// TwinCAT 3 PLC project Twinson
// Title: Twinson
// Company: Stefan Besler
// ProjectVersion: 0.2.0.0
// ProgramVersion: 3.1.4023.0
// project tree:
//   JsonDecoder/ IJsonElement.TcIO, JsonDecoder.TcPOU, JsonElement.TcPOU, JsonElementType.TcDUT, JsonNode.TcDUT
//   JsonDecoder/_Test/ JsonDecoderTest.TcPOU
//   / ParameterList.TcGVL
//   UnitTest/ IAssertions.TcIO, IUnittest.TcIO

// ---- JsonDecoder/JsonElementType.TcDUT
{attribute 'qualified_only'}
TYPE JsonElementType :
(
  Undefined := 0,
  Strng,
  Number,
  Object,
  Arry,
  Boolean,
  Null
);
END_TYPE

// ---- JsonDecoder/JsonNode.TcDUT
TYPE JsonNode :
STRUCT
  Name : STRING;
  Next : REFERENCE TO JsonNode;
  Child : REFERENCE TO JsonNode;
  Element : REFERENCE TO JsonElement;
END_STRUCT
END_TYPE

// ---- ParameterList.TcGVL
{attribute 'qualified_only'}
VAR_GLOBAL CONSTANT
  MaxJsonKeyLength : INT := 31;
  MaxJsonAssignments : INT := 200;
END_VAR

// ---- JsonDecoder/IJsonElement.TcIO
INTERFACE IJsonElement

METHOD AsString : STRING
END_METHOD

END_INTERFACE

// ---- UnitTest/IAssertions.TcIO
/// see [Zeugwerk Unittest](https://doc.zeugwerk.dev/reference/ZCore/UnitTest/IAssertions.html)
INTERFACE IAssertions

/// Asserts that two STRINGs are equal. If they are not, an assertion error is created.
METHOD PUBLIC EqualsString
VAR_INPUT
  expected : STRING(255); //< STRING expected value
  actual : STRING(255); //< STRING actual value
  message : STRING(255); // The identifying message for the assertion error
END_VAR
END_METHOD

/// Asserts that a condition is false. If it is not, an assertion error is created.
METHOD PUBLIC IsFalse
VAR_INPUT
  condition : BOOL; //< Condition to be checked
  message : STRING(255); //< The identifying message for the assertion error
END_VAR
END_METHOD

/// Asserts that a condition is true. If it is not, an assertion error is created.
METHOD PUBLIC IsTrue
VAR_INPUT
  condition : BOOL; //< Condition to be checked
  message : STRING(255); //< The identifying message for the assertion error
END_VAR
END_METHOD

END_INTERFACE

// ---- UnitTest/IUnittest.TcIO
/// see [Zeugwerk Unittest](https://doc.zeugwerk.dev/reference/ZCore/UnitTest/IUnitTest.html)
INTERFACE IUnittest

END_INTERFACE

// ---- JsonDecoder/JsonDecoder.TcPOU
{attribute 'conditionalshow_all_locals'}
{attribute 'no_explicit_call' := 'JsonDecoder is a class, do not call'}
FUNCTION_BLOCK JsonDecoder
VAR
  _key : STRING;
  _jsonPtr : POINTER TO BYTE;
  _memPtr : POINTER TO BYTE;
  
  _elements : ARRAY[0..ParameterList.MaxJsonAssignments] OF JsonElement;
  _elementCount : UINT;  
  
  _root : JsonNode;
  _nodes : ARRAY[0..ParameterList.MaxJsonAssignments] OF JsonNode;
  _nodeCount : UINT;
  
  _el : JsonElementType;
END_VAR
VAR_OUTPUT
  Error : BOOL;
  ErrorMessage : STRING;
END_VAR

METHOD PROTECTED _Element : IJsonElement
VAR_INPUT
  node : REFERENCE TO JsonNode;
  readPtr : POINTER TO BYTE;
END_VAR
VAR // TEMP
  writePtr : POINTER TO BYTE;
  next : BOOL;
END_VAR
next := TRUE;
node REF= node.Child;
WHILE __ISVALIDREF(node)
DO
  IF next
  THEN
    next := FALSE;
    writePtr := ADR(_key);
    WHILE readPtr^ <> 16#2E AND_THEN readPtr^ <> 16#5B AND_THEN readPtr^ <> 16#5D AND_THEN readPtr^ <> 16#0 // eof, . or [
    DO
      writePtr^ := readPtr^;
      writePtr := writePtr + 1;
      readPtr := readPtr + 1;
    END_WHILE
    writePtr^ := 0;
    
    IF readPtr^ = 16#5D  // skip ]
    THEN 
      readPtr := readPtr + 1; 
    END_IF
    
    IF readPtr^ = 16#2E // skip .  
    THEN 
      readPtr := readPtr + 1;
    END_IF  
    
    IF readPtr^ = 16#5B  // skip [  
    THEN 
      readPtr := readPtr + 1;  
    END_IF  
	END_IF

  IF node.Name = _key
  THEN
    IF readPtr^ <> 0
    THEN
      node REF= node.Child;
      next := TRUE;
    ELSIF __ISVALIDREF(node.Element) // direct access, exact match
    THEN
      _Element := node.Element;
      RETURN;
    END_IF
  ELSE
    node REF= node.Next;    
	END_IF

END_WHILE
END_METHOD

METHOD PROTECTED Abort
VAR_IN_OUT CONSTANT
  errorMessage : STRING;
END_VAR
THIS^.ErrorMessage := errorMessage;
THIS^.Error := TRUE;
END_METHOD

METHOD PROTECTED AddElement
VAR_INPUT
  node : REFERENCE TO JsonNode;
END_VAR
VAR
  element : REFERENCE TO JsonElement;
END_VAR
element REF= _elements[_elementCount];
element.ValueType := _el;
element.StartPtr := _memPtr;
element.EndPtr := _jsonPtr;
_elementCount := _elementCount + 1;

node.Element REF= element;
END_METHOD

METHOD PROTECTED AddNode : REFERENCE TO JsonNode
VAR_INPUT
  node : REFERENCE TO JsonNode;
END_VAR
VAR
  namePtr : POINTER TO BYTE;
  memPtr : POINTER TO BYTE;
END_VAR
AddNode REF= _nodes[_nodeCount];
IF __ISVALIDREF(node.Child)
THEN
  AddNode.Next REF= node.Child;
  node.Child REF= AddNode;
ELSE
  node.Child REF= AddNode;
END_IF

// set node name
namePtr := ADR(AddNode.Name);
memPtr := _memPtr;
WHILE memPtr <> _jsonPtr
DO
  namePtr^ := memPtr^;
  namePtr := namePtr + 1;
  memPtr := memPtr + 1;
END_WHILE
namePtr^ := 0;
// reset elements
AddNode.Child REF= 0;
_nodeCount := _nodeCount + 1;
END_METHOD

METHOD Decode
VAR_IN_OUT CONSTANT
  json : STRING;
END_VAR
_jsonPtr := ADR(json);
_elementCount := 0;
_nodeCount := 0;

Error := FALSE;

WHILE _jsonPtr^ <> 0
DO
  SkipWhitespaces();

  CASE GuessElementType()
  OF
    JsonElementType.Object:
      ParseObject(_root);
    JsonElementType.Arry:
      _memPtr := _jsonPtr;
      _root.Child REF= AddNode(_root);
      _root.Child.Name := 'array';
      ParseArray(_root.Child);
  ELSE
    Abort('Unexpected character');
    RETURN;
	END_CASE
  
  _jsonPtr := _jsonPtr + 1;
END_WHILE
END_METHOD

METHOD Element : IJsonElement
VAR_IN_OUT CONSTANT
  path : STRING;
END_VAR
Element := _Element(_root, ADR(path));
END_METHOD

METHOD PROTECTED GuessElementType : JsonElementType
CASE _jsonPtr^
OF
  16#22: // "
    GuessElementType := JsonElementType.Strng;
  16#30..16#39, // 0-9
  16#2B, // +
  16#2D, // -
  16#2E, // .
  16#65, // e
  16#45: // E
    GuessElementType := JsonElementType.Number;    
  16#7B: // {
    GuessElementType := JsonElementType.Object;
  16#5B: // [
    GuessElementType := JsonElementType.Arry;
  16#66, // f
  16#74: // t
    GuessElementType := JsonElementType.Boolean;
  16#6E: // n
    GuessElementType := JsonElementType.Null;      
END_CASE
END_METHOD

METHOD PROTECTED IntToString
VAR_INPUT
  element : INT;
END_VAR
VAR_IN_OUT CONSTANT
  str : STRING;
END_VAR
VAR
  writePtr : POINTER TO BYTE;
  reversePtr : POINTER TO BYTE;  
  endPtr : POINTER TO BYTE;  
END_VAR
writePtr := ADR(str);

// for ints below ten, conversion is easy
IF element < 10
THEN
  writePtr^ := 16#30 + INT_TO_BYTE(element);
  writePtr[1] := 0;
  RETURN;
END_IF

// for more elements it gets trickier
// we have to write the index in reverse, for element 12, we first build a string
// that looks like 21 and then we reverse it, because we apriori don't know how many
// characters will come
REPEAT
  writePtr^ := INT_TO_BYTE(element MOD 10) + 16#30; writePtr := writePtr + 1;
  element := element / 10; 
UNTIL element = 0 END_REPEAT
writePtr^ := 0;

// reverse string with XOR swap algorithm
reversePtr := ADR(str);
endPtr := writePtr - 1;
WHILE reversePtr < endPtr
DO
  // swap first and last
  reversePtr^ := endPtr^ XOR reversePtr^;
  endPtr^ := reversePtr^ XOR endPtr^;
  reversePtr^ := endPtr^ XOR reversePtr^;
  
  reversePtr := reversePtr + 1;
  endPtr := endPtr - 1;
END_WHILE
END_METHOD

METHOD PROTECTED ParseArray
VAR_INPUT
  node : REFERENCE TO JsonNode;
END_VAR
VAR
  child : REFERENCE TO JsonNode;
  elements : INT;
END_VAR
_jsonPtr := _jsonPtr + 1;

REPEAT

  _memPtr := _jsonPtr; // we set the name by index later on
  child REF= AddNode(node);
  IntToString(elements, child.Name);
  elements := elements + 1;
  ParseElement(child);
  
  // got another element in this object?
  IF _jsonPtr^ = 16#2C // ,
  THEN
    _jsonPtr := _jsonPtr + 1; // ,
    SkipWhitespaces();      
  END_IF    

UNTIL _jsonPtr^ = 16#5D OR_ELSE _jsonPtr^ = 0 END_REPEAT // } or EOF

IF _jsonPtr^ <> 0
THEN
  // skip ]
  _jsonPtr := _jsonPtr + 1;
END_IF
END_METHOD

METHOD PROTECTED ParseElement
VAR_INPUT
  node : REFERENCE TO JsonNode;  
END_VAR
VAR
  child : REFERENCE TO JsonNode;
END_VAR
SkipWhitespaces();
_el := GuessElementType();
CASE _el
OF
  JsonElementType.Strng:
    // skip " and additional whitespaces
    _jsonPtr := _jsonPtr + 1;
    _memPtr := _jsonPtr;
    SkipString();
    AddElement(node);
    // skip "
    _jsonPtr := _jsonPtr + 1;    
  
  JsonElementType.Number:
    _memPtr := _jsonPtr;
    SkipNumber();
    AddElement(node);
    
  JsonElementType.Object:
    ParseObject(node);
  
  JsonElementType.Arry:
    ParseArray(node);
    
  JsonElementType.Boolean:
    _memPtr := _jsonPtr;
    SkipBoolean();
    AddElement(node);
    
  JsonElementType.Null:
    _memPtr := _jsonPtr;
    _jsonPtr := _jsonPtr + 4; // null
    AddElement(node);
ELSE
  Abort('Unexpected character');
  RETURN;
END_CASE
SkipWhitespaces();
END_METHOD

METHOD PROTECTED ParseObject
VAR_INPUT
  node : REFERENCE TO JsonNode;  
END_VAR
VAR
  child : REFERENCE TO JsonNode;
  childNamePtr : POINTER TO BYTE;
END_VAR
// skip {
_jsonPtr := _jsonPtr + 1;
SkipWhitespaces();

REPEAT

  _el := GuessElementType();
  IF _el <> JsonElementType.Strng
  THEN
    Abort('Unexpected character');
    RETURN;    
  END_IF
  
  // skip "
  _jsonPtr := _jsonPtr + 1;
  _memPtr := _jsonPtr;
  SkipString();
  
  // chain key
  child REF= AddNode(node);
    
  // skip " and additional whitespaces
  _jsonPtr := _jsonPtr + 1;
  SkipWhitespaces();
  
  IF _jsonPtr^ <> 16#3A // :
  THEN
    Abort('Expected colon');
    RETURN;
  END_IF
  
  // skip :
  _jsonPtr := _jsonPtr + 1;
  ParseElement(child);
  
  // got another element in this object?
  IF _jsonPtr^ = 16#2C // ,
  THEN
    _jsonPtr := _jsonPtr + 1; // ,
    SkipWhitespaces();      
  END_IF  
  
UNTIL _jsonPtr^ = 16#7D OR_ELSE _jsonPtr^ = 0 END_REPEAT // } or EOF

IF _jsonPtr^ <> 0
THEN
  // skip }
  _jsonPtr := _jsonPtr + 1;
END_IF
END_METHOD

METHOD PROTECTED SkipBoolean
IF _jsonPtr^ = 16#66 // f
THEN
  _jsonPtr := _jsonPtr + 1; // false
END_IF

_jsonPtr := _jsonPtr + 4; // true
END_METHOD

METHOD PROTECTED SkipNumber
WHILE (_jsonPtr^ >= 16#30 AND_THEN _jsonPtr^ <= 16#39) OR_ELSE _jsonPtr^ = 16#2B OR_ELSE _jsonPtr^ = 16#2D OR_ELSE _jsonPtr^ = 16#2E OR_ELSE _jsonPtr^ = 16#65 OR_ELSE _jsonPtr^ = 16#45
DO
  _jsonPtr := _jsonPtr + 1;
END_WHILE
END_METHOD

METHOD PROTECTED SkipString
WHILE _jsonPtr^ <> 16#22
DO
  _jsonPtr := _jsonPtr + 1;
END_WHILE
END_METHOD

METHOD PROTECTED SkipWhitespaces
WHILE _jsonPtr^ > 0 AND_THEN _jsonPtr^ <= 16#20
DO
  _jsonPtr := _jsonPtr + 1;
END_WHILE
END_METHOD

END_FUNCTION_BLOCK

// ---- JsonDecoder/JsonElement.TcPOU
FUNCTION_BLOCK JsonElement IMPLEMENTS IJsonElement
VAR_INPUT
  StartPtr : POINTER TO BYTE;
  EndPtr : POINTER TO BYTE;
  ValueType : JsonElementType;
END_VAR

METHOD AsString : STRING
VAR
  it : POINTER TO BYTE;
  retrn : POINTER TO BYTE;  
END_VAR
it := StartPtr;
retrn := ADR(AsString);
WHILE it <> EndPtr
DO
  retrn^ := it^;
  retrn := retrn + 1;
  it := it + 1;
END_WHILE

retrn^ := 0;
END_METHOD

END_FUNCTION_BLOCK

// ---- JsonDecoder/_Test/JsonDecoderTest.TcPOU
FUNCTION_BLOCK JsonDecoderTest EXTENDS JsonDecoder IMPLEMENTS IUnitTest

METHOD Test_Decode_NestedArray
VAR_INPUT
  assertions : IAssertions;
END_VAR
VAR
  element0 : IJsonElement;
  element1 : IJsonElement;
  element2 : IJsonElement;  
END_VAR
Decode('[[[4,2,3]]]');
element0 := Element('array[0][0][0]');
element1 := Element('array[0][0][1]');
element2 := Element('array[0][0][2]');

assertions.IsTrue(element0 <> 0, '');
assertions.IsTrue(element1 <> 0, '');
assertions.IsTrue(element2 <> 0, '');

IF element0 <> 0 AND element1 <> 0 AND element2 <> 0
THEN
	assertions.EqualsString('4', element0.AsString(), '');
	assertions.EqualsString('2', element1.AsString(), '');
	assertions.EqualsString('3', element2.AsString(), '');
END_IF
END_METHOD

METHOD Test_IntToString
VAR_INPUT
  assertions : IAssertions;
END_VAR
VAR
  str : STRING;
END_VAR
str := '';
IntToString(0, str);
assertions.EqualsString(expected := '0', actual := str, message:='Index 0 is correctly converted to an array index key');

str := '';
IntToString(1, str);
assertions.EqualsString(expected := '1', actual := str, message:='Index 1 is correctly converted to an array index key');

str := '';
IntToString(9, str);
assertions.EqualsString(expected := '9', actual := str, message:='Index 9 is correctly converted to an array index key');

str := '';
IntToString(10, str);
assertions.EqualsString(expected := '10', actual := str, message:='Index 10 is correctly converted to an array index key');

str := '';
IntToString(55, str);
assertions.EqualsString(expected := '55', actual := str, message:='Index 55 is correctly converted to an array index key');
END_METHOD

METHOD Test_SkipWhitespace
VAR_INPUT
  assertions : IAssertions;
END_VAR
VAR
  json : STRING;  
END_VAR
json := '              

        !';
_jsonPtr := ADR(json);
SkipWhitespaces();

_jsonPtr^ := 16#33;
END_METHOD

END_FUNCTION_BLOCK
